// LS Electric XG5000 project: SPAV_PANEL
// PLC LSPLC
// module base 0 slot 0: 입출력 모듈:XBC-DN/DP30E (DC 24V 입력 18점, 트랜지스터 출력 12점)

PROGRAM 00MAIN (task: 占쏙옙캔 占쏙옙占싸그뤄옙)

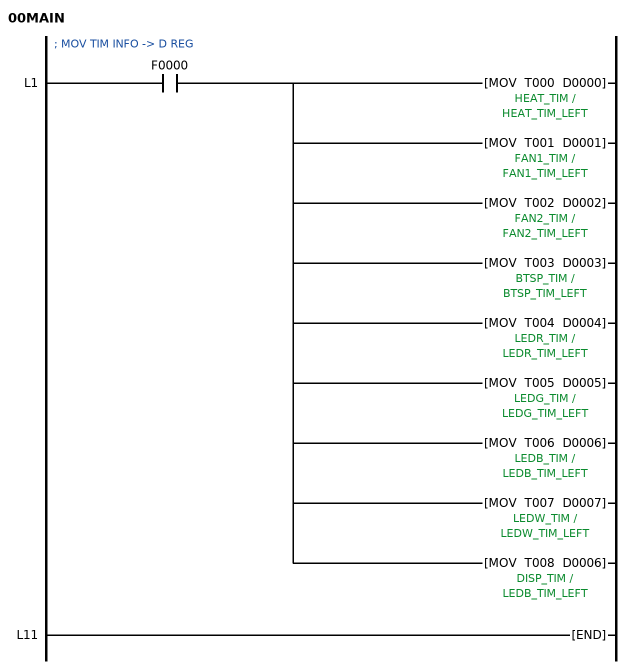
// MOV TIM INFO -> D REG
; L1
LOAD      F0000
MOV       T000 D0000	// HEAT_TIM / HEAT_TIM_LEFT
MOV       T001 D0001	// FAN1_TIM / FAN1_TIM_LEFT
MOV       T002 D0002	// FAN2_TIM / FAN2_TIM_LEFT
MOV       T003 D0003	// BTSP_TIM / BTSP_TIM_LEFT
MOV       T004 D0004	// LEDR_TIM / LEDR_TIM_LEFT
MOV       T005 D0005	// LEDG_TIM / LEDG_TIM_LEFT
MOV       T006 D0006	// LEDB_TIM / LEDB_TIM_LEFT
MOV       T007 D0007	// LEDW_TIM / LEDW_TIM_LEFT
MOV       T008 D0006	// DISP_TIM / LEDB_TIM_LEFT
; L11
END

PROGRAM 01INPUT (task: 占쏙옙캔 占쏙옙占싸그뤄옙)

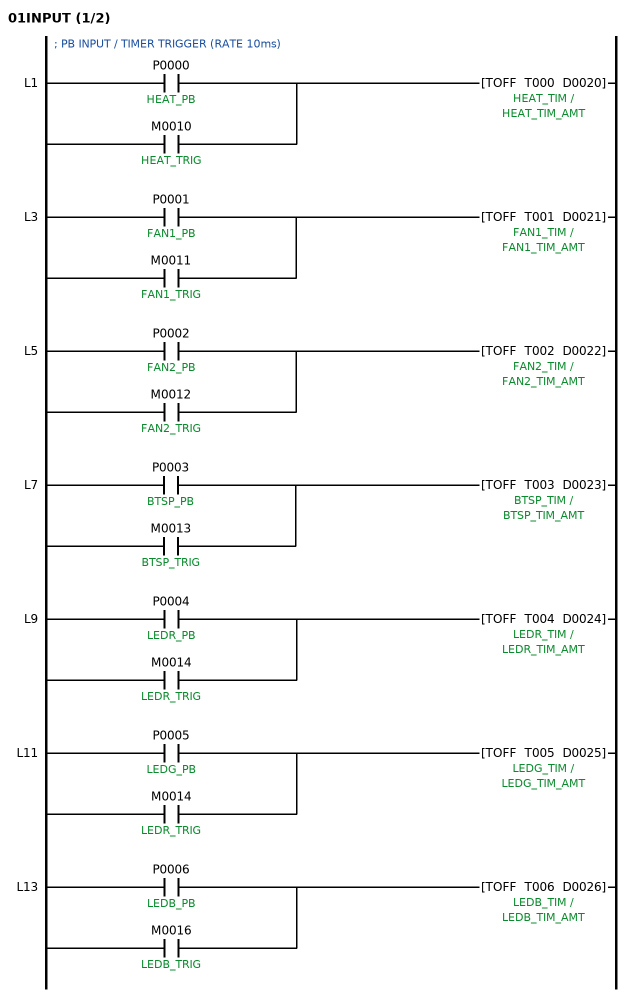
// PB INPUT / TIMER TRIGGER (RATE 10ms)
; L1
LOAD      P0000	// HEAT_PB
OR        M0010	// HEAT_TRIG
TOFF      T000 D0020	// HEAT_TIM / HEAT_TIM_AMT
; L3
LOAD      P0001	// FAN1_PB
OR        M0011	// FAN1_TRIG
TOFF      T001 D0021	// FAN1_TIM / FAN1_TIM_AMT
; L5
LOAD      P0002	// FAN2_PB
OR        M0012	// FAN2_TRIG
TOFF      T002 D0022	// FAN2_TIM / FAN2_TIM_AMT
; L7
LOAD      P0003	// BTSP_PB
OR        M0013	// BTSP_TRIG
TOFF      T003 D0023	// BTSP_TIM / BTSP_TIM_AMT
; L9
LOAD      P0004	// LEDR_PB
OR        M0014	// LEDR_TRIG
TOFF      T004 D0024	// LEDR_TIM / LEDR_TIM_AMT
; L11
LOAD      P0005	// LEDG_PB
OR        M0014	// LEDR_TRIG
TOFF      T005 D0025	// LEDG_TIM / LEDG_TIM_AMT
; L13
LOAD      P0006	// LEDB_PB
OR        M0016	// LEDB_TRIG
TOFF      T006 D0026	// LEDB_TIM / LEDB_TIM_AMT

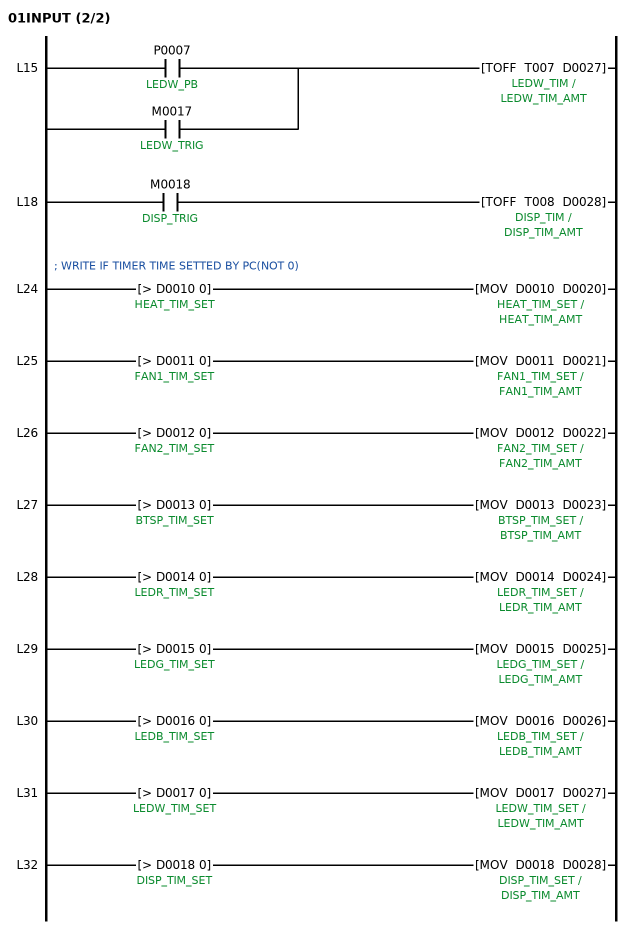
; L15
LOAD      P0007	// LEDW_PB
OR        M0017	// LEDW_TRIG
TOFF      T007 D0027	// LEDW_TIM / LEDW_TIM_AMT
; L18
LOAD      M0018	// DISP_TRIG
TOFF      T008 D0028	// DISP_TIM / DISP_TIM_AMT
// WRITE IF TIMER TIME SETTED BY PC(NOT 0)
; L24
LOAD>     D0010 0	// HEAT_TIM_SET
MOV       D0010 D0020	// HEAT_TIM_SET / HEAT_TIM_AMT
; L25
LOAD>     D0011 0	// FAN1_TIM_SET
MOV       D0011 D0021	// FAN1_TIM_SET / FAN1_TIM_AMT
; L26
LOAD>     D0012 0	// FAN2_TIM_SET
MOV       D0012 D0022	// FAN2_TIM_SET / FAN2_TIM_AMT
; L27
LOAD>     D0013 0	// BTSP_TIM_SET
MOV       D0013 D0023	// BTSP_TIM_SET / BTSP_TIM_AMT
; L28
LOAD>     D0014 0	// LEDR_TIM_SET
MOV       D0014 D0024	// LEDR_TIM_SET / LEDR_TIM_AMT
; L29
LOAD>     D0015 0	// LEDG_TIM_SET
MOV       D0015 D0025	// LEDG_TIM_SET / LEDG_TIM_AMT
; L30
LOAD>     D0016 0	// LEDB_TIM_SET
MOV       D0016 D0026	// LEDB_TIM_SET / LEDB_TIM_AMT
; L31
LOAD>     D0017 0	// LEDW_TIM_SET
MOV       D0017 D0027	// LEDW_TIM_SET / LEDW_TIM_AMT
; L32
LOAD>     D0018 0	// DISP_TIM_SET
MOV       D0018 D0028	// DISP_TIM_SET / DISP_TIM_AMT

PROGRAM 02OUTPUT (task: 占쏙옙캔 占쏙옙占싸그뤄옙)

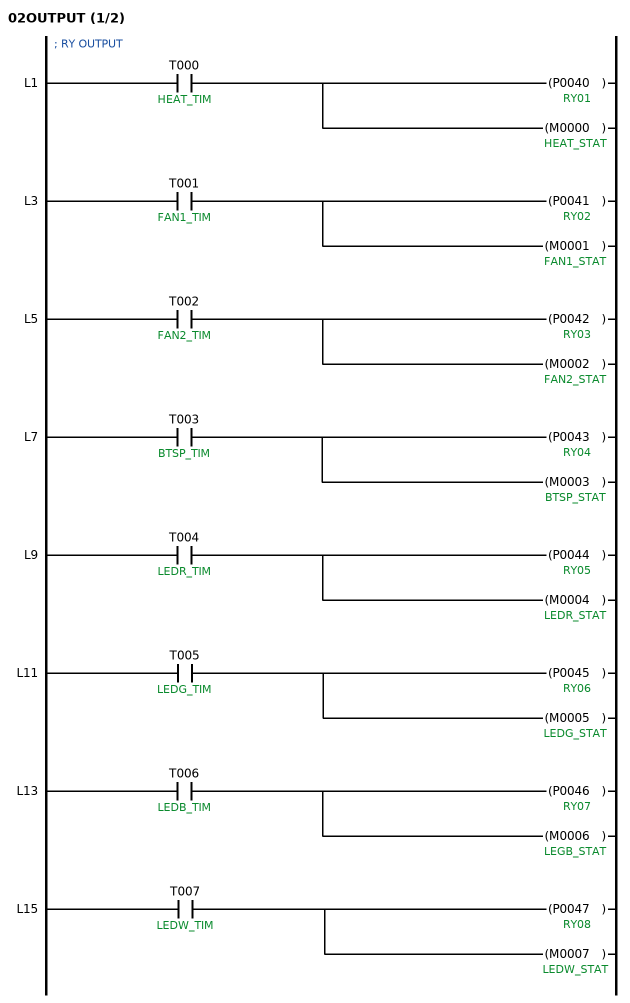
// RY OUTPUT
; L1
LOAD      T000	// HEAT_TIM
OUT       P0040	// RY01
OUT       M0000	// HEAT_STAT
; L3
LOAD      T001	// FAN1_TIM
OUT       P0041	// RY02
OUT       M0001	// FAN1_STAT
; L5
LOAD      T002	// FAN2_TIM
OUT       P0042	// RY03
OUT       M0002	// FAN2_STAT
; L7
LOAD      T003	// BTSP_TIM
OUT       P0043	// RY04
OUT       M0003	// BTSP_STAT
; L9
LOAD      T004	// LEDR_TIM
OUT       P0044	// RY05
OUT       M0004	// LEDR_STAT
; L11
LOAD      T005	// LEDG_TIM
OUT       P0045	// RY06
OUT       M0005	// LEDG_STAT
; L13
LOAD      T006	// LEDB_TIM
OUT       P0046	// RY07
OUT       M0006	// LEGB_STAT
; L15
LOAD      T007	// LEDW_TIM
OUT       P0047	// RY08
OUT       M0007	// LEDW_STAT

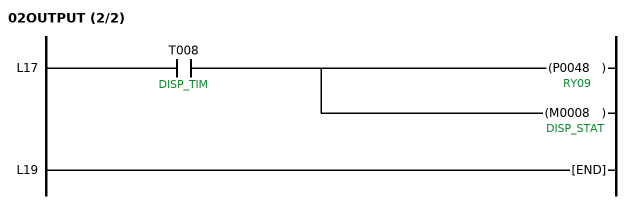
; L17
LOAD      T008	// DISP_TIM
OUT       P0048	// RY09
OUT       M0008	// DISP_STAT
; L19
END

VARIABLES AND COMMENTS (devices not used above)
D00008	WORD	DISP_TIM_LEFT
M00015	BIT	LEDG_TRIG